PROGRAM MAIN
VAR
	// Creation of BOOL variables for button press
	bLeftbutton : BOOL := FALSE;
	bRightbutton: BOOL := FALSE;
	bMachineOn: BOOL := FALSE;
	
	// Here the timer and lockout memory are created
	tTimer: TON;
	bLock: BOOL := FALSE;
END_VAR

// Timer is created with start condtion being if only one button is pressed
tTimer(IN:= bLeftbutton XOR bRightbutton, PT:=T#5S);

//Lock enabled if timer is completed
IF tTimer.Q THEN
	bLock := TRUE;
END_IF;

// Conditional for when both buttons are pressed without Lockout memory being enabled.
IF bLeftbutton AND bRightbutton AND NOT bLock THEN
	bMachineOn := TRUE;
END_IF;

// Final conditional for disabling Lockout when both buttons are not pressed.
IF NOT bLeftbutton AND NOT bRightbutton THEN
	bLock := FALSE;
END_IF

END_PROGRAM

(* stored: Version 1.1.0.1, ProductVersion 3.1.4024.16
   POU MAIN: Id {db8bfc4a-b855-44fc-bdea-39219db874f6}, SpecialFunc None *)
